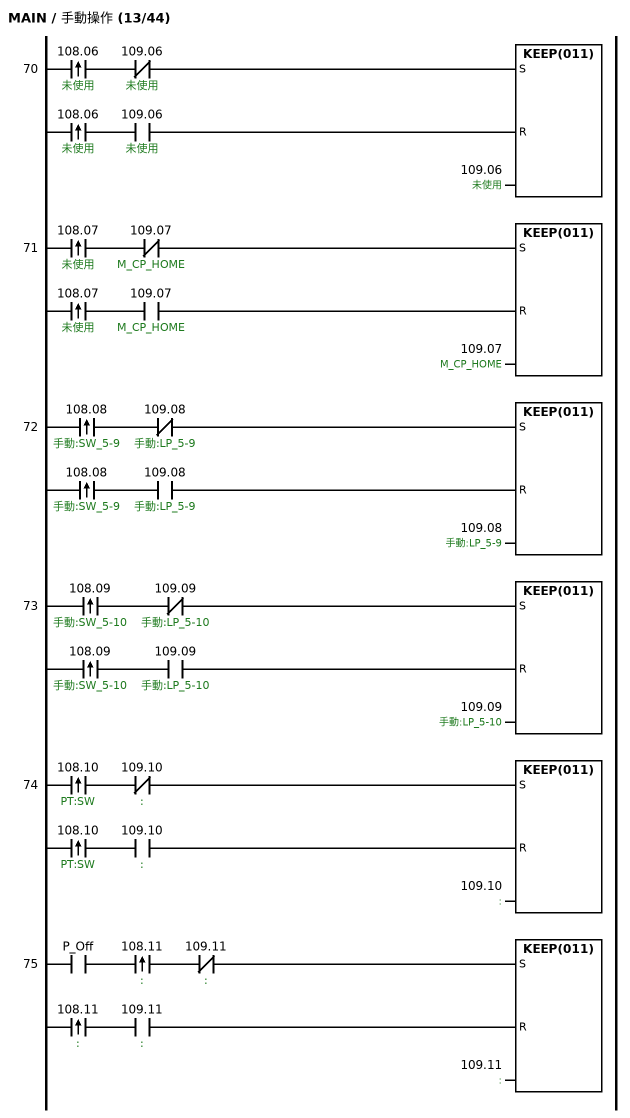
; [picture p48: MAIN / 手動操作, rungs 70-75]
; rung 70
@LD 108.06  ; 未使用
ANDNOT 109.06  ; 未使用
@LD 108.06  ; 未使用
AND 109.06  ; 未使用
KEEP(011) 109.06  ; 未使用
; rung 71
@LD 108.07  ; 未使用
ANDNOT 109.07  ; M_CP_HOME
@LD 108.07  ; 未使用
AND 109.07  ; M_CP_HOME
KEEP(011) 109.07  ; M_CP_HOME
; rung 72
@LD 108.08  ; 手動:SW_5-9
ANDNOT 109.08  ; 手動:LP_5-9
@LD 108.08  ; 手動:SW_5-9
AND 109.08  ; 手動:LP_5-9
KEEP(011) 109.08  ; 手動:LP_5-9
; rung 73
@LD 108.09  ; 手動:SW_5-10
ANDNOT 109.09  ; 手動:LP_5-10
@LD 108.09  ; 手動:SW_5-10
AND 109.09  ; 手動:LP_5-10
KEEP(011) 109.09  ; 手動:LP_5-10
; rung 74
@LD 108.10  ; PT:SW
ANDNOT 109.10  ; :
@LD 108.10  ; PT:SW
AND 109.10  ; :
KEEP(011) 109.10  ; :
; rung 75
LD P_Off
@AND 108.11  ; :
ANDNOT 109.11  ; :
@LD 108.11  ; :
AND 109.11  ; :
KEEP(011) 109.11  ; :

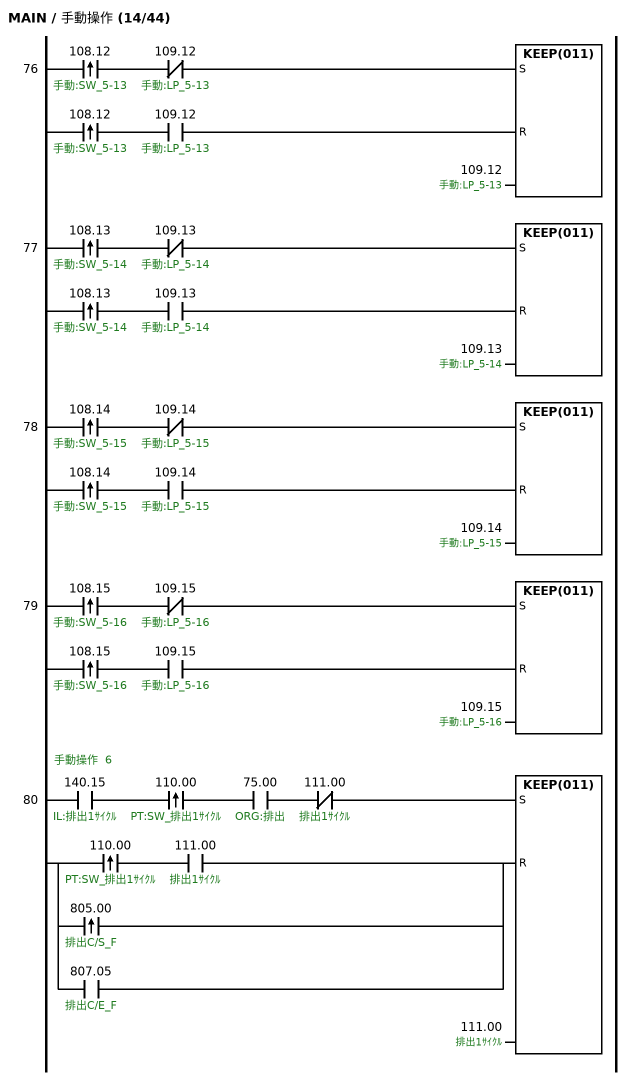
; rung 76
@LD 108.12  ; 手動:SW_5-13
ANDNOT 109.12  ; 手動:LP_5-13
@LD 108.12  ; 手動:SW_5-13
AND 109.12  ; 手動:LP_5-13
KEEP(011) 109.12  ; 手動:LP_5-13
; rung 77
@LD 108.13  ; 手動:SW_5-14
ANDNOT 109.13  ; 手動:LP_5-14
@LD 108.13  ; 手動:SW_5-14
AND 109.13  ; 手動:LP_5-14
KEEP(011) 109.13  ; 手動:LP_5-14
; rung 78
@LD 108.14  ; 手動:SW_5-15
ANDNOT 109.14  ; 手動:LP_5-15
@LD 108.14  ; 手動:SW_5-15
AND 109.14  ; 手動:LP_5-15
KEEP(011) 109.14  ; 手動:LP_5-15
; rung 79
@LD 108.15  ; 手動:SW_5-16
ANDNOT 109.15  ; 手動:LP_5-16
@LD 108.15  ; 手動:SW_5-16
AND 109.15  ; 手動:LP_5-16
KEEP(011) 109.15  ; 手動:LP_5-16
; rung 80: 手動操作  6
LD 140.15  ; IL:排出1ｻｲｸﾙ
@AND 110.00  ; PT:SW_排出1ｻｲｸﾙ
AND 75.00  ; ORG:排出
ANDNOT 111.00  ; 排出1ｻｲｸﾙ
@LD 110.00  ; PT:SW_排出1ｻｲｸﾙ
AND 111.00  ; 排出1ｻｲｸﾙ
@OR 805.00  ; 排出C/S_F
OR 807.05  ; 排出C/E_F
KEEP(011) 111.00  ; 排出1ｻｲｸﾙ

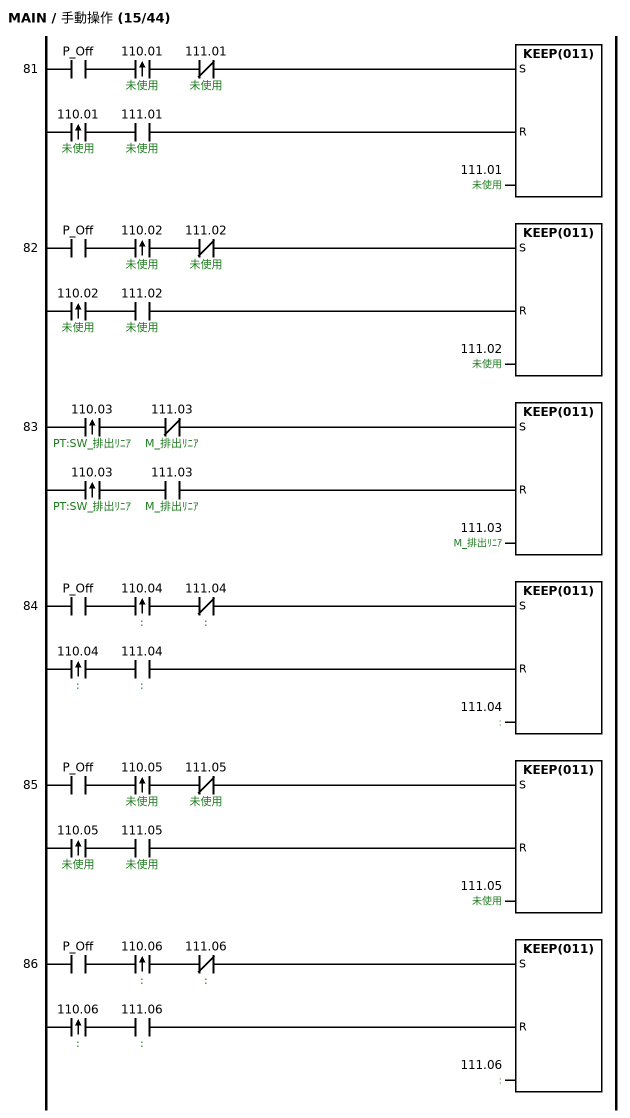
; rung 81
LD P_Off
@AND 110.01  ; 未使用
ANDNOT 111.01  ; 未使用
@LD 110.01  ; 未使用
AND 111.01  ; 未使用
KEEP(011) 111.01  ; 未使用
; rung 82
LD P_Off
@AND 110.02  ; 未使用
ANDNOT 111.02  ; 未使用
@LD 110.02  ; 未使用
AND 111.02  ; 未使用
KEEP(011) 111.02  ; 未使用
; rung 83
@LD 110.03  ; PT:SW_排出ﾘﾆｱ
ANDNOT 111.03  ; M_排出ﾘﾆｱ
@LD 110.03  ; PT:SW_排出ﾘﾆｱ
AND 111.03  ; M_排出ﾘﾆｱ
KEEP(011) 111.03  ; M_排出ﾘﾆｱ
; rung 84
LD P_Off
@AND 110.04  ; :
ANDNOT 111.04  ; :
@LD 110.04  ; :
AND 111.04  ; :
KEEP(011) 111.04  ; :
; rung 85
LD P_Off
@AND 110.05  ; 未使用
ANDNOT 111.05  ; 未使用
@LD 110.05  ; 未使用
AND 111.05  ; 未使用
KEEP(011) 111.05  ; 未使用
; rung 86
LD P_Off
@AND 110.06  ; :
ANDNOT 111.06  ; :
@LD 110.06  ; :
AND 111.06  ; :
KEEP(011) 111.06  ; :

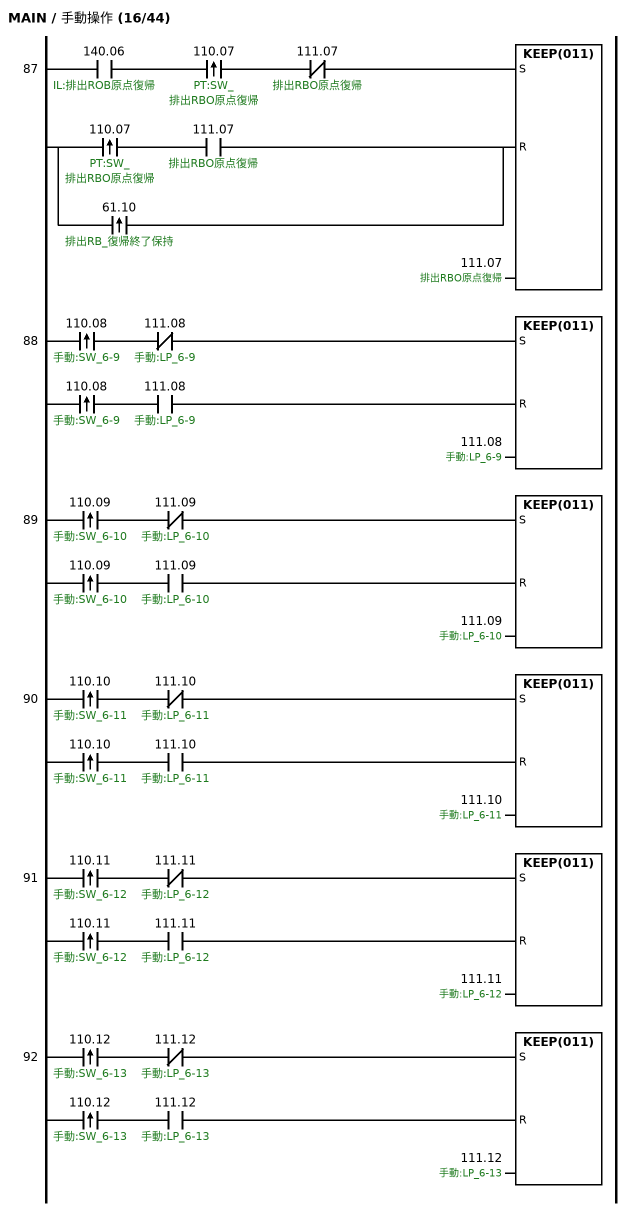
; rung 87
LD 140.06  ; IL:排出ROB原点復帰
@AND 110.07  ; PT:SW_排出RBO原点復帰
ANDNOT 111.07  ; 排出RBO原点復帰
@LD 110.07  ; PT:SW_排出RBO原点復帰
AND 111.07  ; 排出RBO原点復帰
@OR 61.10  ; 排出RB_復帰終了保持
KEEP(011) 111.07  ; 排出RBO原点復帰
; rung 88
@LD 110.08  ; 手動:SW_6-9
ANDNOT 111.08  ; 手動:LP_6-9
@LD 110.08  ; 手動:SW_6-9
AND 111.08  ; 手動:LP_6-9
KEEP(011) 111.08  ; 手動:LP_6-9
; rung 89
@LD 110.09  ; 手動:SW_6-10
ANDNOT 111.09  ; 手動:LP_6-10
@LD 110.09  ; 手動:SW_6-10
AND 111.09  ; 手動:LP_6-10
KEEP(011) 111.09  ; 手動:LP_6-10
; rung 90
@LD 110.10  ; 手動:SW_6-11
ANDNOT 111.10  ; 手動:LP_6-11
@LD 110.10  ; 手動:SW_6-11
AND 111.10  ; 手動:LP_6-11
KEEP(011) 111.10  ; 手動:LP_6-11
; rung 91
@LD 110.11  ; 手動:SW_6-12
ANDNOT 111.11  ; 手動:LP_6-12
@LD 110.11  ; 手動:SW_6-12
AND 111.11  ; 手動:LP_6-12
KEEP(011) 111.11  ; 手動:LP_6-12
; rung 92
@LD 110.12  ; 手動:SW_6-13
ANDNOT 111.12  ; 手動:LP_6-13
@LD 110.12  ; 手動:SW_6-13
AND 111.12  ; 手動:LP_6-13
KEEP(011) 111.12  ; 手動:LP_6-13

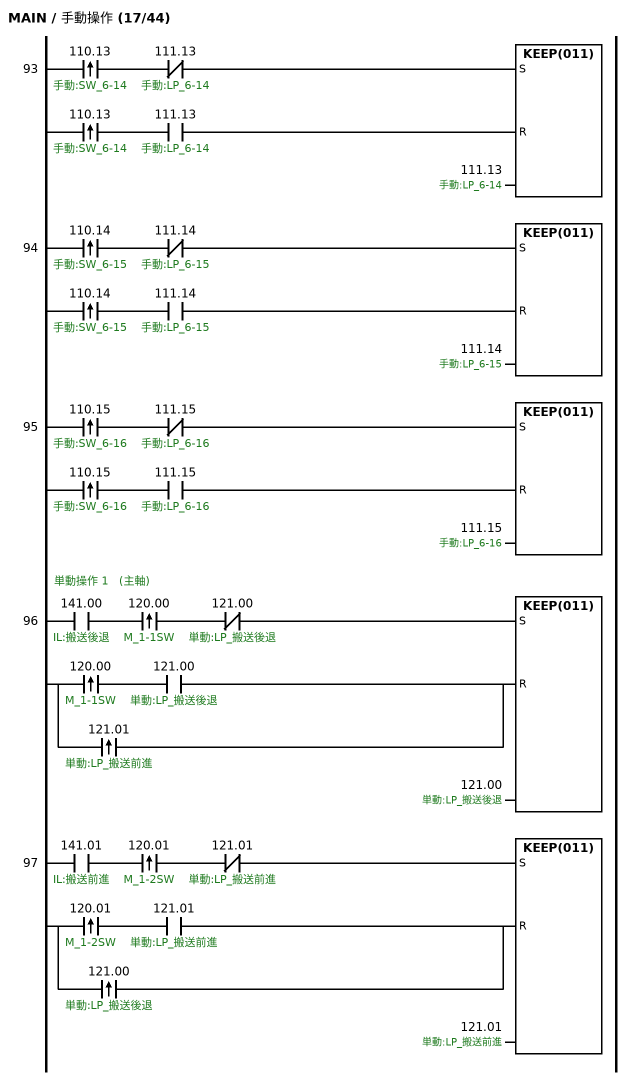
; rung 93
@LD 110.13  ; 手動:SW_6-14
ANDNOT 111.13  ; 手動:LP_6-14
@LD 110.13  ; 手動:SW_6-14
AND 111.13  ; 手動:LP_6-14
KEEP(011) 111.13  ; 手動:LP_6-14
; rung 94
@LD 110.14  ; 手動:SW_6-15
ANDNOT 111.14  ; 手動:LP_6-15
@LD 110.14  ; 手動:SW_6-15
AND 111.14  ; 手動:LP_6-15
KEEP(011) 111.14  ; 手動:LP_6-15
; rung 95
@LD 110.15  ; 手動:SW_6-16
ANDNOT 111.15  ; 手動:LP_6-16
@LD 110.15  ; 手動:SW_6-16
AND 111.15  ; 手動:LP_6-16
KEEP(011) 111.15  ; 手動:LP_6-16
; rung 96: 単動操作 1   (主軸)
LD 141.00  ; IL:搬送後退
@AND 120.00  ; M_1-1SW
ANDNOT 121.00  ; 単動:LP_搬送後退
@LD 120.00  ; M_1-1SW
AND 121.00  ; 単動:LP_搬送後退
@OR 121.01  ; 単動:LP_搬送前進
KEEP(011) 121.00  ; 単動:LP_搬送後退
; rung 97
LD 141.01  ; IL:搬送前進
@AND 120.01  ; M_1-2SW
ANDNOT 121.01  ; 単動:LP_搬送前進
@LD 120.01  ; M_1-2SW
AND 121.01  ; 単動:LP_搬送前進
@OR 121.00  ; 単動:LP_搬送後退
KEEP(011) 121.01  ; 単動:LP_搬送前進

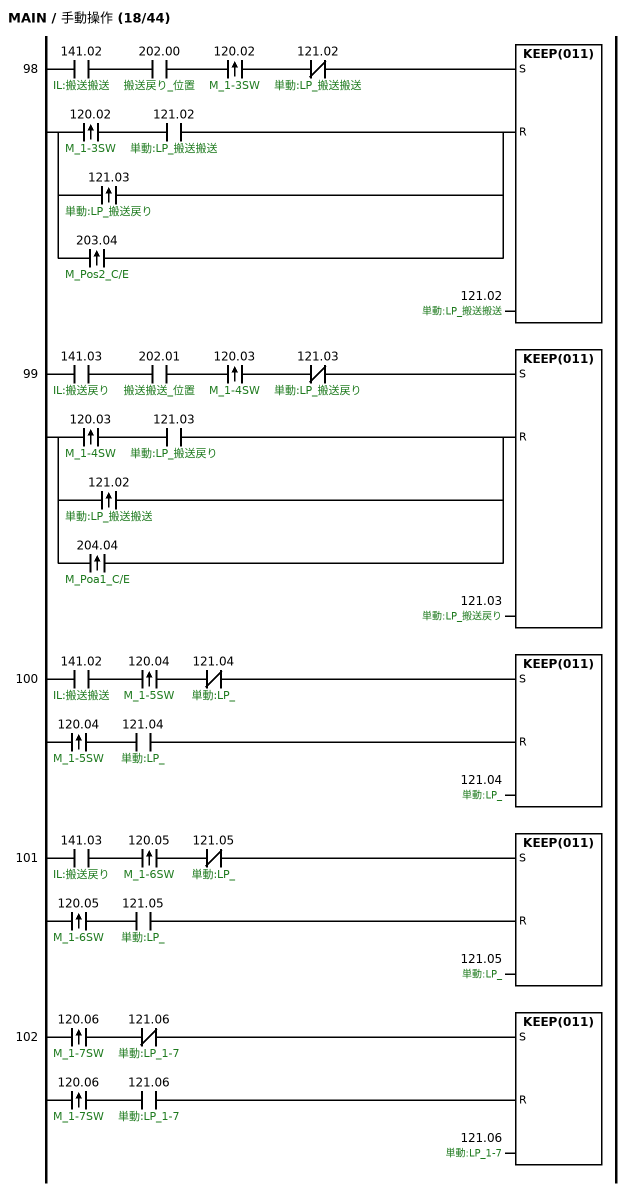
; rung 98
LD 141.02  ; IL:搬送搬送
AND 202.00  ; 搬送戻り_位置
@AND 120.02  ; M_1-3SW
ANDNOT 121.02  ; 単動:LP_搬送搬送
@LD 120.02  ; M_1-3SW
AND 121.02  ; 単動:LP_搬送搬送
@OR 121.03  ; 単動:LP_搬送戻り
@OR 203.04  ; M_Pos2_C/E
KEEP(011) 121.02  ; 単動:LP_搬送搬送
; rung 99
LD 141.03  ; IL:搬送戻り
AND 202.01  ; 搬送搬送_位置
@AND 120.03  ; M_1-4SW
ANDNOT 121.03  ; 単動:LP_搬送戻り
@LD 120.03  ; M_1-4SW
AND 121.03  ; 単動:LP_搬送戻り
@OR 121.02  ; 単動:LP_搬送搬送
@OR 204.04  ; M_Poa1_C/E
KEEP(011) 121.03  ; 単動:LP_搬送戻り
; rung 100
LD 141.02  ; IL:搬送搬送
@AND 120.04  ; M_1-5SW
ANDNOT 121.04  ; 単動:LP_
@LD 120.04  ; M_1-5SW
AND 121.04  ; 単動:LP_
KEEP(011) 121.04  ; 単動:LP_
; rung 101
LD 141.03  ; IL:搬送戻り
@AND 120.05  ; M_1-6SW
ANDNOT 121.05  ; 単動:LP_
@LD 120.05  ; M_1-6SW
AND 121.05  ; 単動:LP_
KEEP(011) 121.05  ; 単動:LP_
; rung 102
@LD 120.06  ; M_1-7SW
ANDNOT 121.06  ; 単動:LP_1-7
@LD 120.06  ; M_1-7SW
AND 121.06  ; 単動:LP_1-7
KEEP(011) 121.06  ; 単動:LP_1-7

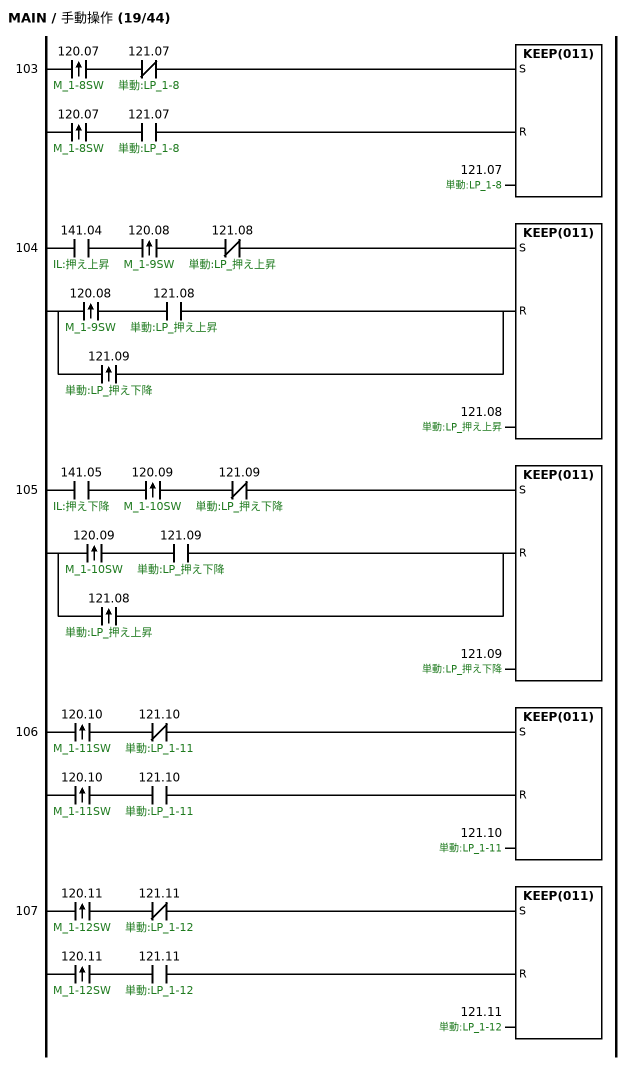
; rung 103
@LD 120.07  ; M_1-8SW
ANDNOT 121.07  ; 単動:LP_1-8
@LD 120.07  ; M_1-8SW
AND 121.07  ; 単動:LP_1-8
KEEP(011) 121.07  ; 単動:LP_1-8
; rung 104
LD 141.04  ; IL:押え上昇
@AND 120.08  ; M_1-9SW
ANDNOT 121.08  ; 単動:LP_押え上昇
@LD 120.08  ; M_1-9SW
AND 121.08  ; 単動:LP_押え上昇
@OR 121.09  ; 単動:LP_押え下降
KEEP(011) 121.08  ; 単動:LP_押え上昇
; rung 105
LD 141.05  ; IL:押え下降
@AND 120.09  ; M_1-10SW
ANDNOT 121.09  ; 単動:LP_押え下降
@LD 120.09  ; M_1-10SW
AND 121.09  ; 単動:LP_押え下降
@OR 121.08  ; 単動:LP_押え上昇
KEEP(011) 121.09  ; 単動:LP_押え下降
; rung 106
@LD 120.10  ; M_1-11SW
ANDNOT 121.10  ; 単動:LP_1-11
@LD 120.10  ; M_1-11SW
AND 121.10  ; 単動:LP_1-11
KEEP(011) 121.10  ; 単動:LP_1-11
; rung 107
@LD 120.11  ; M_1-12SW
ANDNOT 121.11  ; 単動:LP_1-12
@LD 120.11  ; M_1-12SW
AND 121.11  ; 単動:LP_1-12
KEEP(011) 121.11  ; 単動:LP_1-12

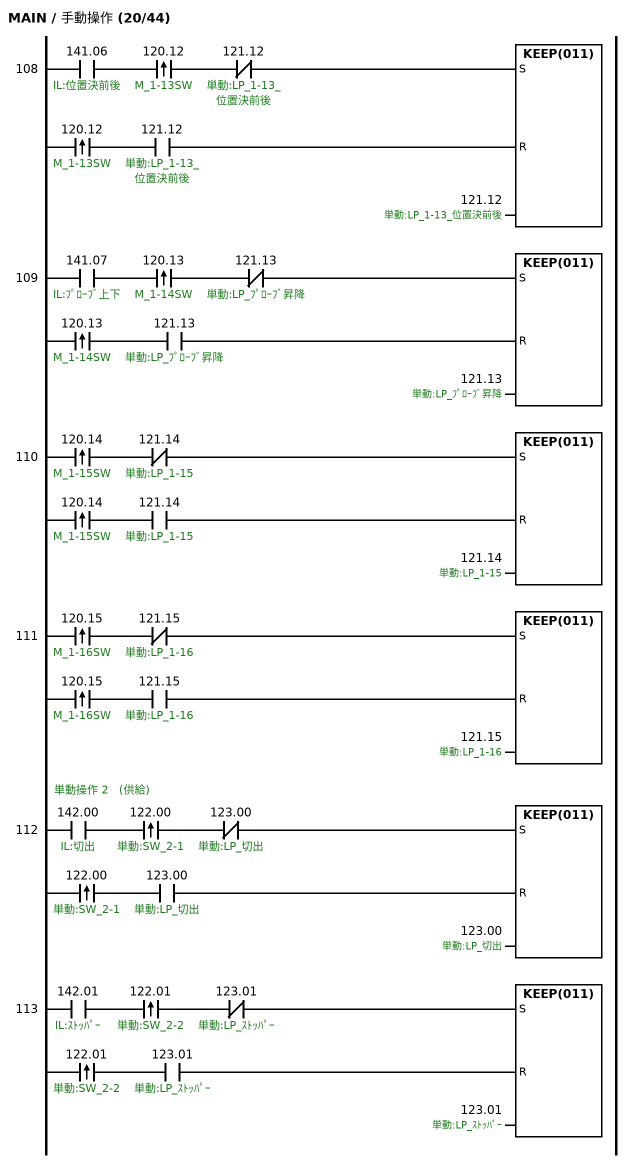
; rung 108
LD 141.06  ; IL:位置決前後
@AND 120.12  ; M_1-13SW
ANDNOT 121.12  ; 単動:LP_1-13_位置決前後
@LD 120.12  ; M_1-13SW
AND 121.12  ; 単動:LP_1-13_位置決前後
KEEP(011) 121.12  ; 単動:LP_1-13_位置決前後
; rung 109
LD 141.07  ; IL:ﾌﾟﾛｰﾌﾞ上下
@AND 120.13  ; M_1-14SW
ANDNOT 121.13  ; 単動:LP_ﾌﾟﾛｰﾌﾞ昇降
@LD 120.13  ; M_1-14SW
AND 121.13  ; 単動:LP_ﾌﾟﾛｰﾌﾞ昇降
KEEP(011) 121.13  ; 単動:LP_ﾌﾟﾛｰﾌﾞ昇降
; rung 110
@LD 120.14  ; M_1-15SW
ANDNOT 121.14  ; 単動:LP_1-15
@LD 120.14  ; M_1-15SW
AND 121.14  ; 単動:LP_1-15
KEEP(011) 121.14  ; 単動:LP_1-15
; rung 111
@LD 120.15  ; M_1-16SW
ANDNOT 121.15  ; 単動:LP_1-16
@LD 120.15  ; M_1-16SW
AND 121.15  ; 単動:LP_1-16
KEEP(011) 121.15  ; 単動:LP_1-16
; rung 112: 単動操作 2   (供給)
LD 142.00  ; IL:切出
@AND 122.00  ; 単動:SW_2-1
ANDNOT 123.00  ; 単動:LP_切出
@LD 122.00  ; 単動:SW_2-1
AND 123.00  ; 単動:LP_切出
KEEP(011) 123.00  ; 単動:LP_切出
; rung 113
LD 142.01  ; IL:ｽﾄｯﾊﾟｰ
@AND 122.01  ; 単動:SW_2-2
ANDNOT 123.01  ; 単動:LP_ｽﾄｯﾊﾟｰ
@LD 122.01  ; 単動:SW_2-2
AND 123.01  ; 単動:LP_ｽﾄｯﾊﾟｰ
KEEP(011) 123.01  ; 単動:LP_ｽﾄｯﾊﾟｰ

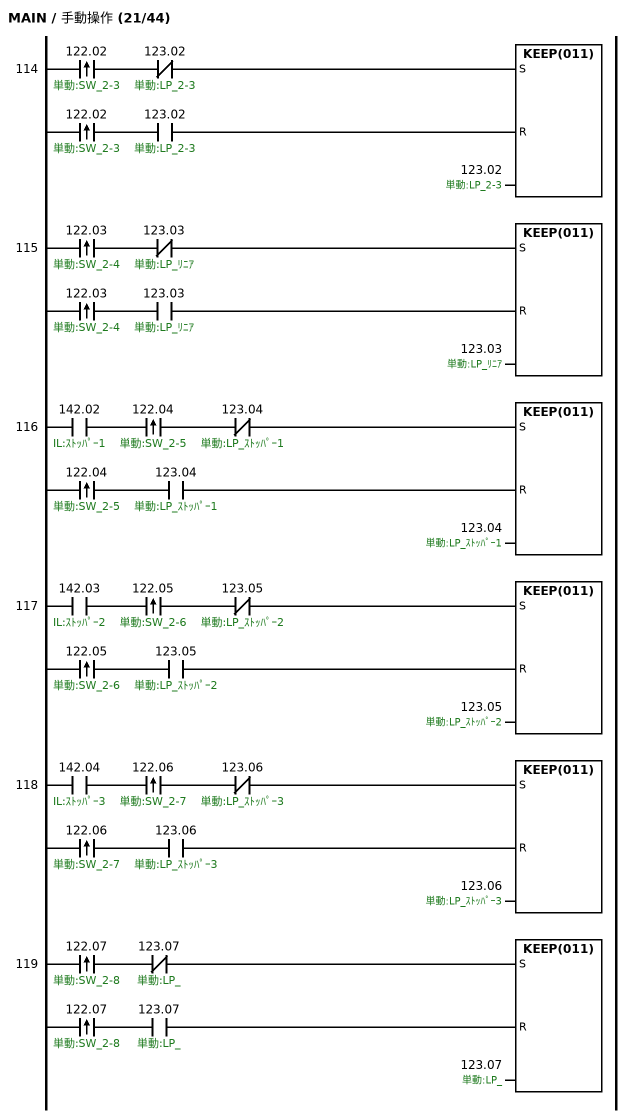
; rung 114
@LD 122.02  ; 単動:SW_2-3
ANDNOT 123.02  ; 単動:LP_2-3
@LD 122.02  ; 単動:SW_2-3
AND 123.02  ; 単動:LP_2-3
KEEP(011) 123.02  ; 単動:LP_2-3
; rung 115
@LD 122.03  ; 単動:SW_2-4
ANDNOT 123.03  ; 単動:LP_ﾘﾆｱ
@LD 122.03  ; 単動:SW_2-4
AND 123.03  ; 単動:LP_ﾘﾆｱ
KEEP(011) 123.03  ; 単動:LP_ﾘﾆｱ
; rung 116
LD 142.02  ; IL:ｽﾄｯﾊﾟｰ1
@AND 122.04  ; 単動:SW_2-5
ANDNOT 123.04  ; 単動:LP_ｽﾄｯﾊﾟｰ1
@LD 122.04  ; 単動:SW_2-5
AND 123.04  ; 単動:LP_ｽﾄｯﾊﾟｰ1
KEEP(011) 123.04  ; 単動:LP_ｽﾄｯﾊﾟｰ1
; rung 117
LD 142.03  ; IL:ｽﾄｯﾊﾟｰ2
@AND 122.05  ; 単動:SW_2-6
ANDNOT 123.05  ; 単動:LP_ｽﾄｯﾊﾟｰ2
@LD 122.05  ; 単動:SW_2-6
AND 123.05  ; 単動:LP_ｽﾄｯﾊﾟｰ2
KEEP(011) 123.05  ; 単動:LP_ｽﾄｯﾊﾟｰ2
; rung 118
LD 142.04  ; IL:ｽﾄｯﾊﾟｰ3
@AND 122.06  ; 単動:SW_2-7
ANDNOT 123.06  ; 単動:LP_ｽﾄｯﾊﾟｰ3
@LD 122.06  ; 単動:SW_2-7
AND 123.06  ; 単動:LP_ｽﾄｯﾊﾟｰ3
KEEP(011) 123.06  ; 単動:LP_ｽﾄｯﾊﾟｰ3
; rung 119
@LD 122.07  ; 単動:SW_2-8
ANDNOT 123.07  ; 単動:LP_
@LD 122.07  ; 単動:SW_2-8
AND 123.07  ; 単動:LP_
KEEP(011) 123.07  ; 単動:LP_

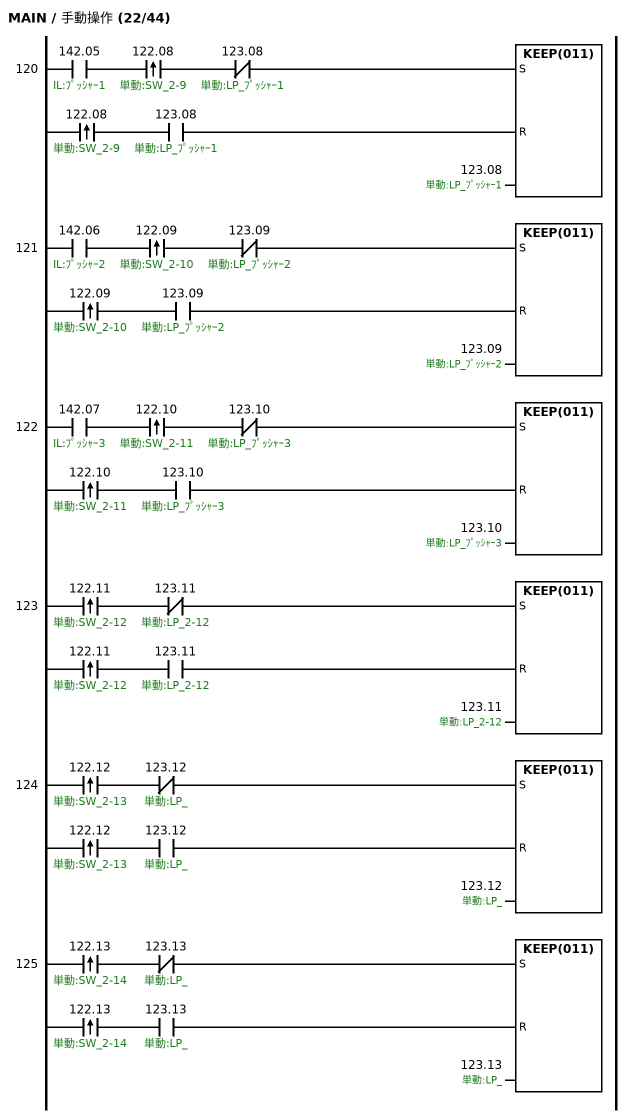
; rung 120
LD 142.05  ; IL:ﾌﾟｯｼｬｰ1
@AND 122.08  ; 単動:SW_2-9
ANDNOT 123.08  ; 単動:LP_ﾌﾟｯｼｬｰ1
@LD 122.08  ; 単動:SW_2-9
AND 123.08  ; 単動:LP_ﾌﾟｯｼｬｰ1
KEEP(011) 123.08  ; 単動:LP_ﾌﾟｯｼｬｰ1
; rung 121
LD 142.06  ; IL:ﾌﾟｯｼｬｰ2
@AND 122.09  ; 単動:SW_2-10
ANDNOT 123.09  ; 単動:LP_ﾌﾟｯｼｬｰ2
@LD 122.09  ; 単動:SW_2-10
AND 123.09  ; 単動:LP_ﾌﾟｯｼｬｰ2
KEEP(011) 123.09  ; 単動:LP_ﾌﾟｯｼｬｰ2
; rung 122
LD 142.07  ; IL:ﾌﾟｯｼｬｰ3
@AND 122.10  ; 単動:SW_2-11
ANDNOT 123.10  ; 単動:LP_ﾌﾟｯｼｬｰ3
@LD 122.10  ; 単動:SW_2-11
AND 123.10  ; 単動:LP_ﾌﾟｯｼｬｰ3
KEEP(011) 123.10  ; 単動:LP_ﾌﾟｯｼｬｰ3
; rung 123
@LD 122.11  ; 単動:SW_2-12
ANDNOT 123.11  ; 単動:LP_2-12
@LD 122.11  ; 単動:SW_2-12
AND 123.11  ; 単動:LP_2-12
KEEP(011) 123.11  ; 単動:LP_2-12
; rung 124
@LD 122.12  ; 単動:SW_2-13
ANDNOT 123.12  ; 単動:LP_
@LD 122.12  ; 単動:SW_2-13
AND 123.12  ; 単動:LP_
KEEP(011) 123.12  ; 単動:LP_
; rung 125
@LD 122.13  ; 単動:SW_2-14
ANDNOT 123.13  ; 単動:LP_
@LD 122.13  ; 単動:SW_2-14
AND 123.13  ; 単動:LP_
KEEP(011) 123.13  ; 単動:LP_

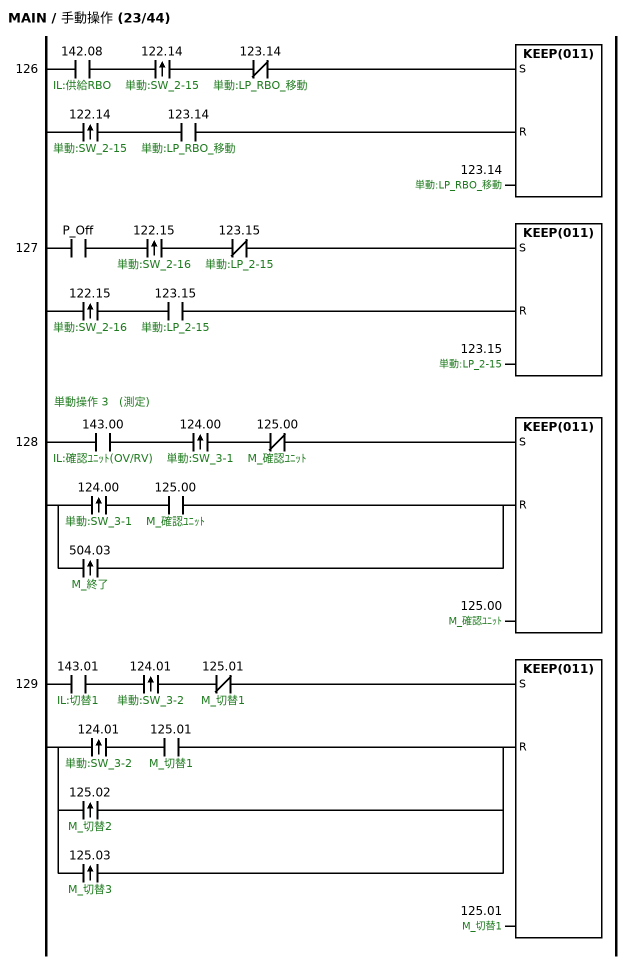
; rung 126
LD 142.08  ; IL:供給RBO
@AND 122.14  ; 単動:SW_2-15
ANDNOT 123.14  ; 単動:LP_RBO_移動
@LD 122.14  ; 単動:SW_2-15
AND 123.14  ; 単動:LP_RBO_移動
KEEP(011) 123.14  ; 単動:LP_RBO_移動
; rung 127
LD P_Off
@AND 122.15  ; 単動:SW_2-16
ANDNOT 123.15  ; 単動:LP_2-15
@LD 122.15  ; 単動:SW_2-16
AND 123.15  ; 単動:LP_2-15
KEEP(011) 123.15  ; 単動:LP_2-15
; rung 128: 単動操作 3   (測定)
LD 143.00  ; IL:確認ﾕﾆｯﾄ(OV/RV)
@AND 124.00  ; 単動:SW_3-1
ANDNOT 125.00  ; M_確認ﾕﾆｯﾄ
@LD 124.00  ; 単動:SW_3-1
AND 125.00  ; M_確認ﾕﾆｯﾄ
@OR 504.03  ; M_終了
KEEP(011) 125.00  ; M_確認ﾕﾆｯﾄ
; rung 129
LD 143.01  ; IL:切替1
@AND 124.01  ; 単動:SW_3-2
ANDNOT 125.01  ; M_切替1
@LD 124.01  ; 単動:SW_3-2
AND 125.01  ; M_切替1
@OR 125.02  ; M_切替2
@OR 125.03  ; M_切替3
KEEP(011) 125.01  ; M_切替1

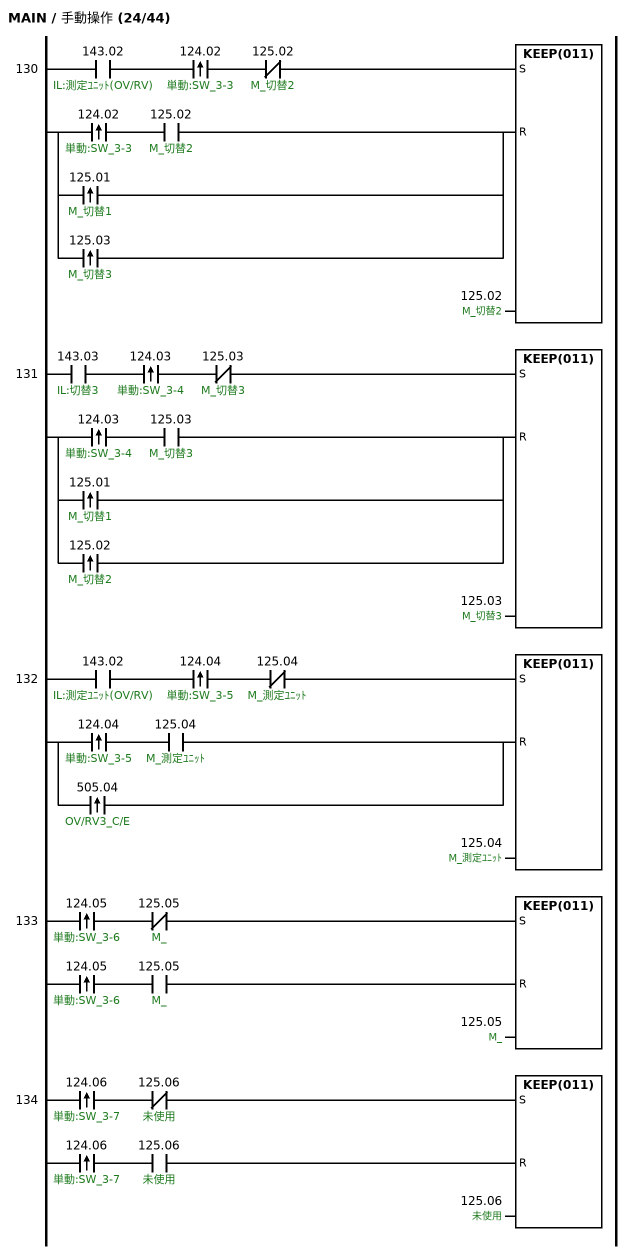
; rung 130
LD 143.02  ; IL:測定ﾕﾆｯﾄ(OV/RV)
@AND 124.02  ; 単動:SW_3-3
ANDNOT 125.02  ; M_切替2
@LD 124.02  ; 単動:SW_3-3
AND 125.02  ; M_切替2
@OR 125.01  ; M_切替1
@OR 125.03  ; M_切替3
KEEP(011) 125.02  ; M_切替2
; rung 131
LD 143.03  ; IL:切替3
@AND 124.03  ; 単動:SW_3-4
ANDNOT 125.03  ; M_切替3
@LD 124.03  ; 単動:SW_3-4
AND 125.03  ; M_切替3
@OR 125.01  ; M_切替1
@OR 125.02  ; M_切替2
KEEP(011) 125.03  ; M_切替3
; rung 132
LD 143.02  ; IL:測定ﾕﾆｯﾄ(OV/RV)
@AND 124.04  ; 単動:SW_3-5
ANDNOT 125.04  ; M_測定ﾕﾆｯﾄ
@LD 124.04  ; 単動:SW_3-5
AND 125.04  ; M_測定ﾕﾆｯﾄ
@OR 505.04  ; OV/RV3_C/E
KEEP(011) 125.04  ; M_測定ﾕﾆｯﾄ
; rung 133
@LD 124.05  ; 単動:SW_3-6
ANDNOT 125.05  ; M_
@LD 124.05  ; 単動:SW_3-6
AND 125.05  ; M_
KEEP(011) 125.05  ; M_
; rung 134
@LD 124.06  ; 単動:SW_3-7
ANDNOT 125.06  ; 未使用
@LD 124.06  ; 単動:SW_3-7
AND 125.06  ; 未使用
KEEP(011) 125.06  ; 未使用

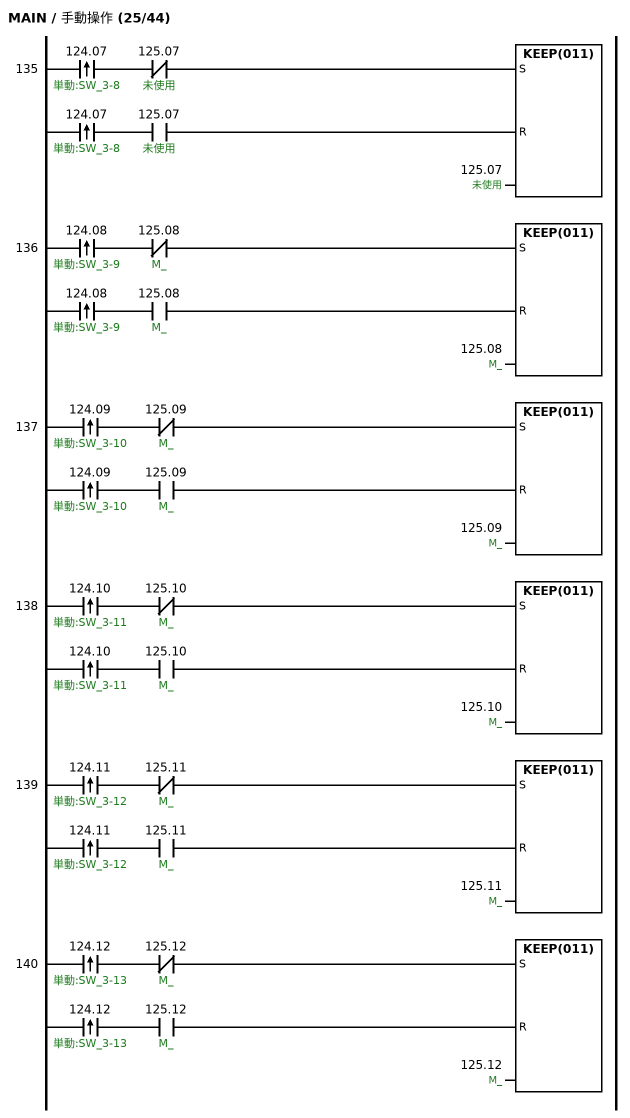
; rung 135
@LD 124.07  ; 単動:SW_3-8
ANDNOT 125.07  ; 未使用
@LD 124.07  ; 単動:SW_3-8
AND 125.07  ; 未使用
KEEP(011) 125.07  ; 未使用
; rung 136
@LD 124.08  ; 単動:SW_3-9
ANDNOT 125.08  ; M_
@LD 124.08  ; 単動:SW_3-9
AND 125.08  ; M_
KEEP(011) 125.08  ; M_
; rung 137
@LD 124.09  ; 単動:SW_3-10
ANDNOT 125.09  ; M_
@LD 124.09  ; 単動:SW_3-10
AND 125.09  ; M_
KEEP(011) 125.09  ; M_
; rung 138
@LD 124.10  ; 単動:SW_3-11
ANDNOT 125.10  ; M_
@LD 124.10  ; 単動:SW_3-11
AND 125.10  ; M_
KEEP(011) 125.10  ; M_
; rung 139
@LD 124.11  ; 単動:SW_3-12
ANDNOT 125.11  ; M_
@LD 124.11  ; 単動:SW_3-12
AND 125.11  ; M_
KEEP(011) 125.11  ; M_
; rung 140
@LD 124.12  ; 単動:SW_3-13
ANDNOT 125.12  ; M_
@LD 124.12  ; 単動:SW_3-13
AND 125.12  ; M_
KEEP(011) 125.12  ; M_

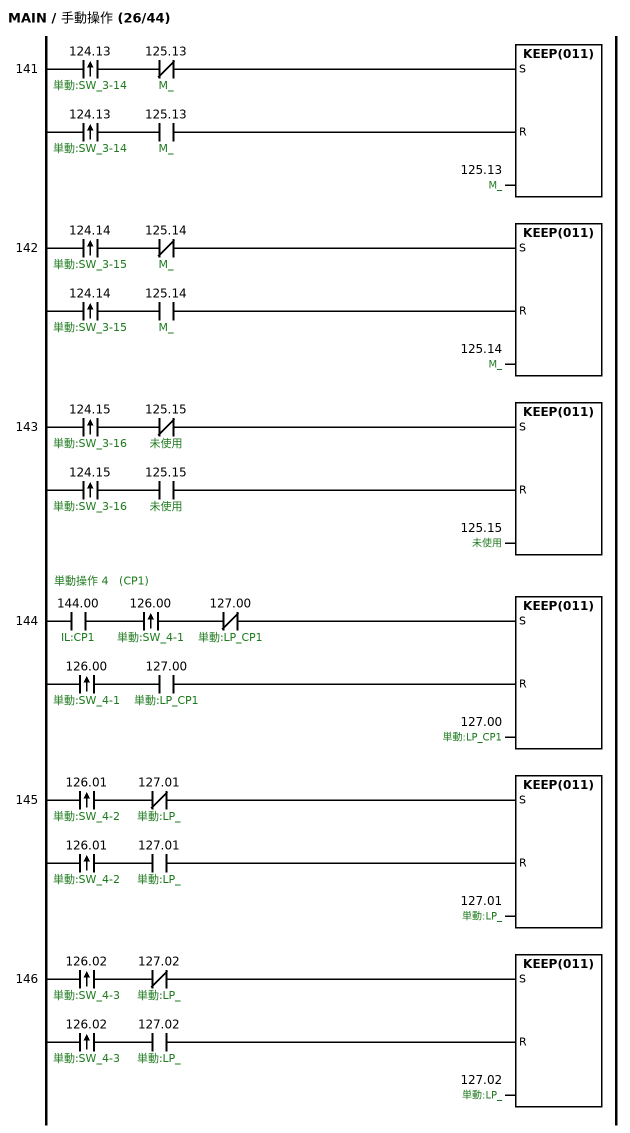
; rung 141
@LD 124.13  ; 単動:SW_3-14
ANDNOT 125.13  ; M_
@LD 124.13  ; 単動:SW_3-14
AND 125.13  ; M_
KEEP(011) 125.13  ; M_
; rung 142
@LD 124.14  ; 単動:SW_3-15
ANDNOT 125.14  ; M_
@LD 124.14  ; 単動:SW_3-15
AND 125.14  ; M_
KEEP(011) 125.14  ; M_
; rung 143
@LD 124.15  ; 単動:SW_3-16
ANDNOT 125.15  ; 未使用
@LD 124.15  ; 単動:SW_3-16
AND 125.15  ; 未使用
KEEP(011) 125.15  ; 未使用
; rung 144: 単動操作 4   (CP1)
LD 144.00  ; IL:CP1
@AND 126.00  ; 単動:SW_4-1
ANDNOT 127.00  ; 単動:LP_CP1
@LD 126.00  ; 単動:SW_4-1
AND 127.00  ; 単動:LP_CP1
KEEP(011) 127.00  ; 単動:LP_CP1
; rung 145
@LD 126.01  ; 単動:SW_4-2
ANDNOT 127.01  ; 単動:LP_
@LD 126.01  ; 単動:SW_4-2
AND 127.01  ; 単動:LP_
KEEP(011) 127.01  ; 単動:LP_
; rung 146
@LD 126.02  ; 単動:SW_4-3
ANDNOT 127.02  ; 単動:LP_
@LD 126.02  ; 単動:SW_4-3
AND 127.02  ; 単動:LP_
KEEP(011) 127.02  ; 単動:LP_

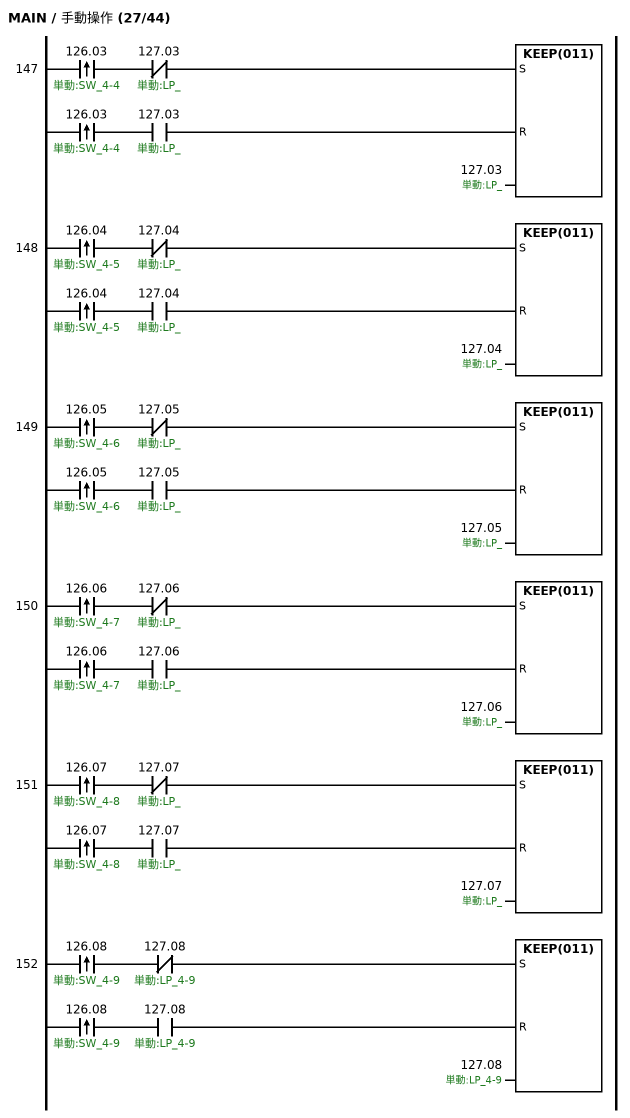
; rung 147
@LD 126.03  ; 単動:SW_4-4
ANDNOT 127.03  ; 単動:LP_
@LD 126.03  ; 単動:SW_4-4
AND 127.03  ; 単動:LP_
KEEP(011) 127.03  ; 単動:LP_
; rung 148
@LD 126.04  ; 単動:SW_4-5
ANDNOT 127.04  ; 単動:LP_
@LD 126.04  ; 単動:SW_4-5
AND 127.04  ; 単動:LP_
KEEP(011) 127.04  ; 単動:LP_
; rung 149
@LD 126.05  ; 単動:SW_4-6
ANDNOT 127.05  ; 単動:LP_
@LD 126.05  ; 単動:SW_4-6
AND 127.05  ; 単動:LP_
KEEP(011) 127.05  ; 単動:LP_
; rung 150
@LD 126.06  ; 単動:SW_4-7
ANDNOT 127.06  ; 単動:LP_
@LD 126.06  ; 単動:SW_4-7
AND 127.06  ; 単動:LP_
KEEP(011) 127.06  ; 単動:LP_
; rung 151
@LD 126.07  ; 単動:SW_4-8
ANDNOT 127.07  ; 単動:LP_
@LD 126.07  ; 単動:SW_4-8
AND 127.07  ; 単動:LP_
KEEP(011) 127.07  ; 単動:LP_
; rung 152
@LD 126.08  ; 単動:SW_4-9
ANDNOT 127.08  ; 単動:LP_4-9
@LD 126.08  ; 単動:SW_4-9
AND 127.08  ; 単動:LP_4-9
KEEP(011) 127.08  ; 単動:LP_4-9

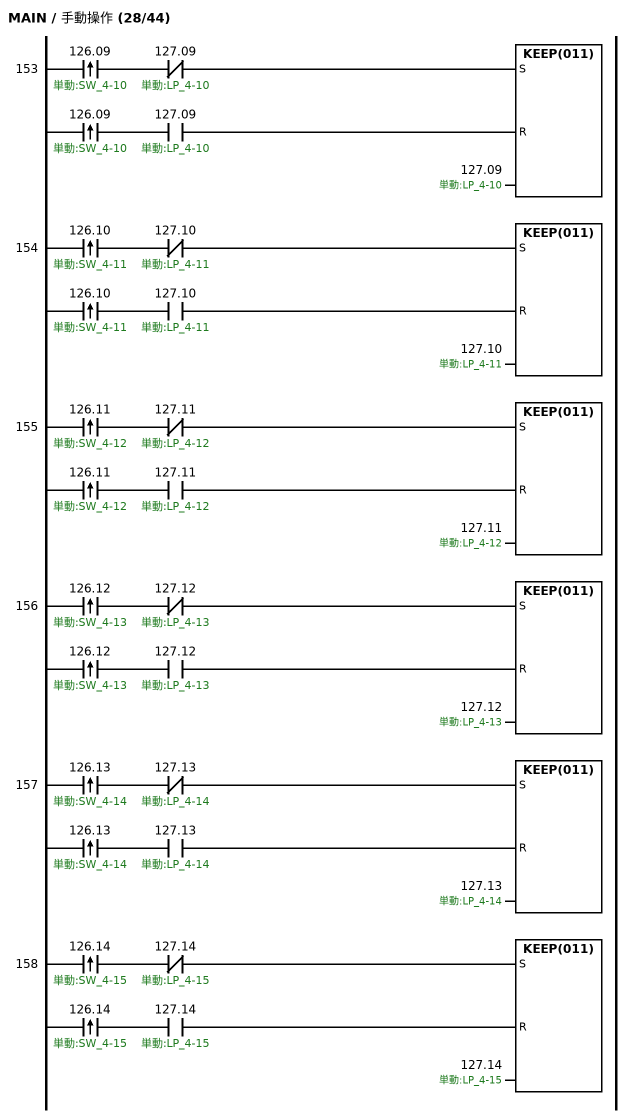
; rung 153
@LD 126.09  ; 単動:SW_4-10
ANDNOT 127.09  ; 単動:LP_4-10
@LD 126.09  ; 単動:SW_4-10
AND 127.09  ; 単動:LP_4-10
KEEP(011) 127.09  ; 単動:LP_4-10
; rung 154
@LD 126.10  ; 単動:SW_4-11
ANDNOT 127.10  ; 単動:LP_4-11
@LD 126.10  ; 単動:SW_4-11
AND 127.10  ; 単動:LP_4-11
KEEP(011) 127.10  ; 単動:LP_4-11
; rung 155
@LD 126.11  ; 単動:SW_4-12
ANDNOT 127.11  ; 単動:LP_4-12
@LD 126.11  ; 単動:SW_4-12
AND 127.11  ; 単動:LP_4-12
KEEP(011) 127.11  ; 単動:LP_4-12
; rung 156
@LD 126.12  ; 単動:SW_4-13
ANDNOT 127.12  ; 単動:LP_4-13
@LD 126.12  ; 単動:SW_4-13
AND 127.12  ; 単動:LP_4-13
KEEP(011) 127.12  ; 単動:LP_4-13
; rung 157
@LD 126.13  ; 単動:SW_4-14
ANDNOT 127.13  ; 単動:LP_4-14
@LD 126.13  ; 単動:SW_4-14
AND 127.13  ; 単動:LP_4-14
KEEP(011) 127.13  ; 単動:LP_4-14
; rung 158
@LD 126.14  ; 単動:SW_4-15
ANDNOT 127.14  ; 単動:LP_4-15
@LD 126.14  ; 単動:SW_4-15
AND 127.14  ; 単動:LP_4-15
KEEP(011) 127.14  ; 単動:LP_4-15

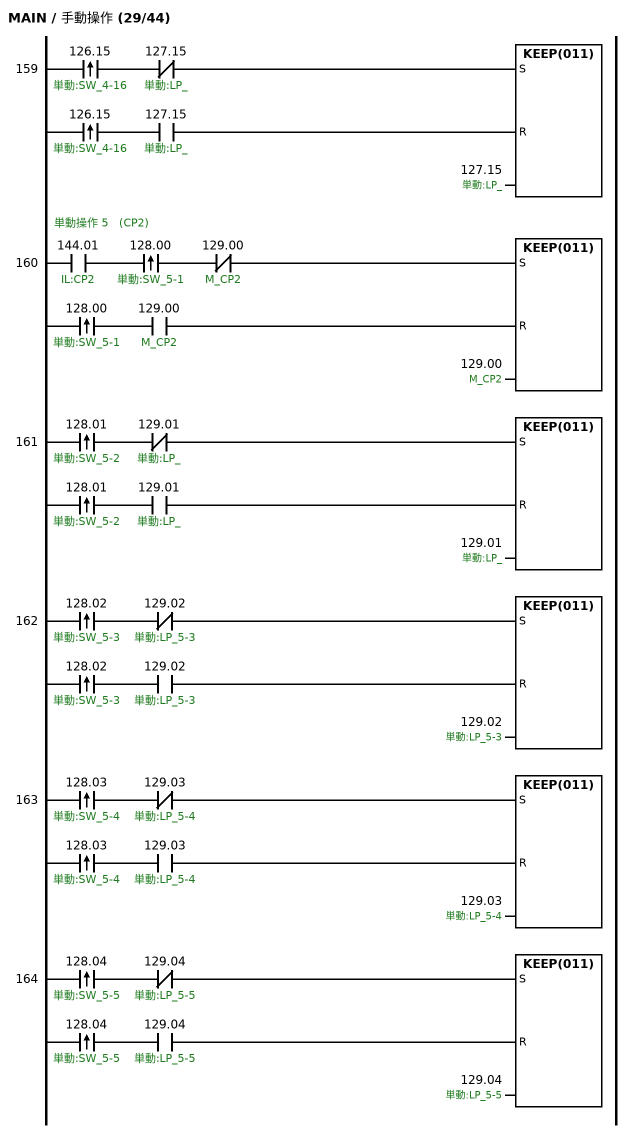
; rung 159
@LD 126.15  ; 単動:SW_4-16
ANDNOT 127.15  ; 単動:LP_
@LD 126.15  ; 単動:SW_4-16
AND 127.15  ; 単動:LP_
KEEP(011) 127.15  ; 単動:LP_
; rung 160: 単動操作 5   (CP2)
LD 144.01  ; IL:CP2
@AND 128.00  ; 単動:SW_5-1
ANDNOT 129.00  ; M_CP2
@LD 128.00  ; 単動:SW_5-1
AND 129.00  ; M_CP2
KEEP(011) 129.00  ; M_CP2
; rung 161
@LD 128.01  ; 単動:SW_5-2
ANDNOT 129.01  ; 単動:LP_
@LD 128.01  ; 単動:SW_5-2
AND 129.01  ; 単動:LP_
KEEP(011) 129.01  ; 単動:LP_
; rung 162
@LD 128.02  ; 単動:SW_5-3
ANDNOT 129.02  ; 単動:LP_5-3
@LD 128.02  ; 単動:SW_5-3
AND 129.02  ; 単動:LP_5-3
KEEP(011) 129.02  ; 単動:LP_5-3
; rung 163
@LD 128.03  ; 単動:SW_5-4
ANDNOT 129.03  ; 単動:LP_5-4
@LD 128.03  ; 単動:SW_5-4
AND 129.03  ; 単動:LP_5-4
KEEP(011) 129.03  ; 単動:LP_5-4
; rung 164
@LD 128.04  ; 単動:SW_5-5
ANDNOT 129.04  ; 単動:LP_5-5
@LD 128.04  ; 単動:SW_5-5
AND 129.04  ; 単動:LP_5-5
KEEP(011) 129.04  ; 単動:LP_5-5

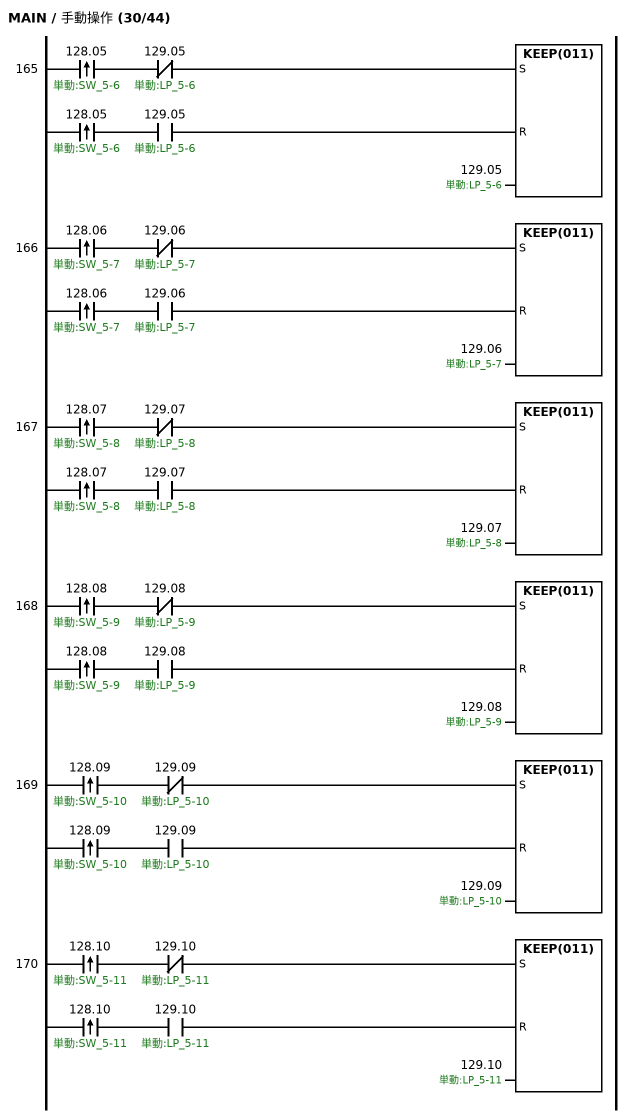
; rung 165
@LD 128.05  ; 単動:SW_5-6
ANDNOT 129.05  ; 単動:LP_5-6
@LD 128.05  ; 単動:SW_5-6
AND 129.05  ; 単動:LP_5-6
KEEP(011) 129.05  ; 単動:LP_5-6
; rung 166
@LD 128.06  ; 単動:SW_5-7
ANDNOT 129.06  ; 単動:LP_5-7
@LD 128.06  ; 単動:SW_5-7
AND 129.06  ; 単動:LP_5-7
KEEP(011) 129.06  ; 単動:LP_5-7
; rung 167
@LD 128.07  ; 単動:SW_5-8
ANDNOT 129.07  ; 単動:LP_5-8
@LD 128.07  ; 単動:SW_5-8
AND 129.07  ; 単動:LP_5-8
KEEP(011) 129.07  ; 単動:LP_5-8
; rung 168
@LD 128.08  ; 単動:SW_5-9
ANDNOT 129.08  ; 単動:LP_5-9
@LD 128.08  ; 単動:SW_5-9
AND 129.08  ; 単動:LP_5-9
KEEP(011) 129.08  ; 単動:LP_5-9
; rung 169
@LD 128.09  ; 単動:SW_5-10
ANDNOT 129.09  ; 単動:LP_5-10
@LD 128.09  ; 単動:SW_5-10
AND 129.09  ; 単動:LP_5-10
KEEP(011) 129.09  ; 単動:LP_5-10
; rung 170
@LD 128.10  ; 単動:SW_5-11
ANDNOT 129.10  ; 単動:LP_5-11
@LD 128.10  ; 単動:SW_5-11
AND 129.10  ; 単動:LP_5-11
KEEP(011) 129.10  ; 単動:LP_5-11

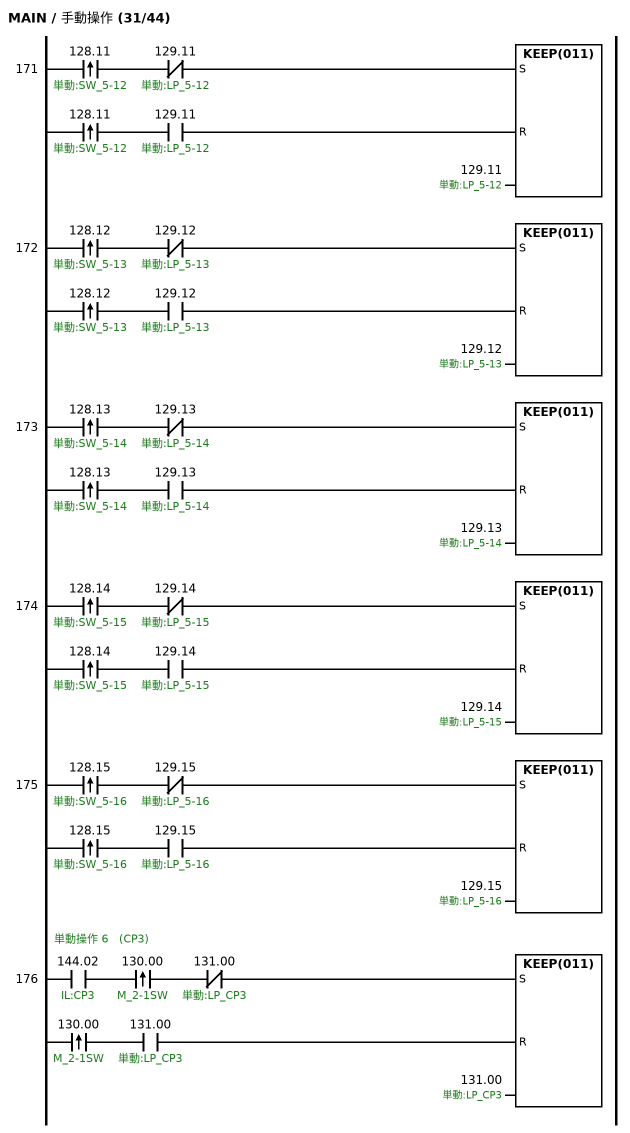
; rung 171
@LD 128.11  ; 単動:SW_5-12
ANDNOT 129.11  ; 単動:LP_5-12
@LD 128.11  ; 単動:SW_5-12
AND 129.11  ; 単動:LP_5-12
KEEP(011) 129.11  ; 単動:LP_5-12
; rung 172
@LD 128.12  ; 単動:SW_5-13
ANDNOT 129.12  ; 単動:LP_5-13
@LD 128.12  ; 単動:SW_5-13
AND 129.12  ; 単動:LP_5-13
KEEP(011) 129.12  ; 単動:LP_5-13
; rung 173
@LD 128.13  ; 単動:SW_5-14
ANDNOT 129.13  ; 単動:LP_5-14
@LD 128.13  ; 単動:SW_5-14
AND 129.13  ; 単動:LP_5-14
KEEP(011) 129.13  ; 単動:LP_5-14
; rung 174
@LD 128.14  ; 単動:SW_5-15
ANDNOT 129.14  ; 単動:LP_5-15
@LD 128.14  ; 単動:SW_5-15
AND 129.14  ; 単動:LP_5-15
KEEP(011) 129.14  ; 単動:LP_5-15
; rung 175
@LD 128.15  ; 単動:SW_5-16
ANDNOT 129.15  ; 単動:LP_5-16
@LD 128.15  ; 単動:SW_5-16
AND 129.15  ; 単動:LP_5-16
KEEP(011) 129.15  ; 単動:LP_5-16
; rung 176: 単動操作 6   (CP3)
LD 144.02  ; IL:CP3
@AND 130.00  ; M_2-1SW
ANDNOT 131.00  ; 単動:LP_CP3
@LD 130.00  ; M_2-1SW
AND 131.00  ; 単動:LP_CP3
KEEP(011) 131.00  ; 単動:LP_CP3

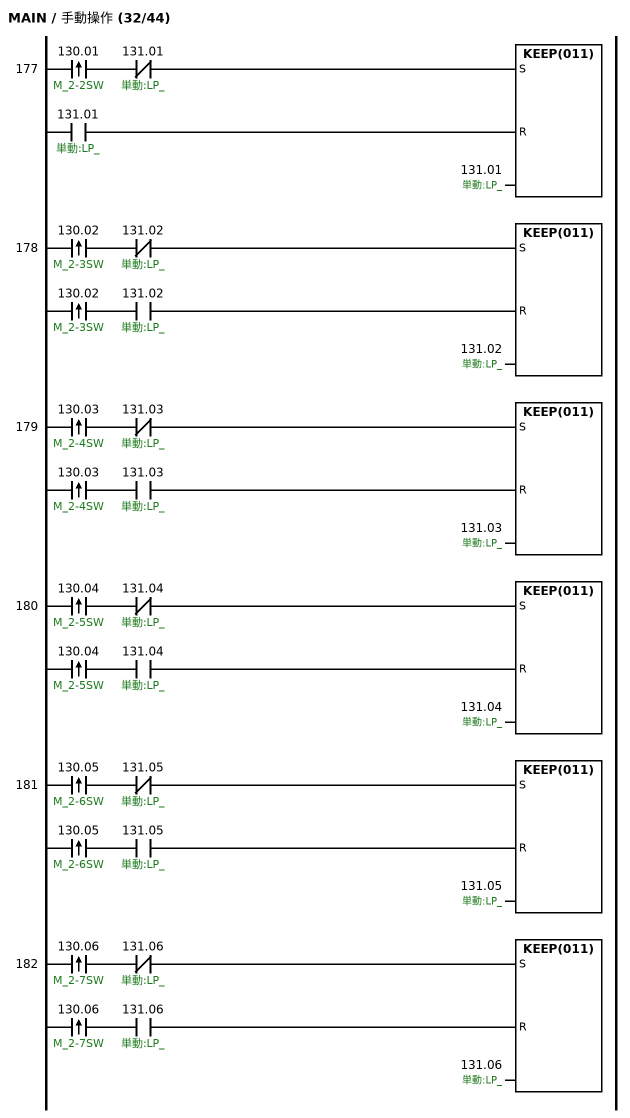
; rung 177
@LD 130.01  ; M_2-2SW
ANDNOT 131.01  ; 単動:LP_
LD 131.01  ; 単動:LP_
KEEP(011) 131.01  ; 単動:LP_
; rung 178
@LD 130.02  ; M_2-3SW
ANDNOT 131.02  ; 単動:LP_
@LD 130.02  ; M_2-3SW
AND 131.02  ; 単動:LP_
KEEP(011) 131.02  ; 単動:LP_
; rung 179
@LD 130.03  ; M_2-4SW
ANDNOT 131.03  ; 単動:LP_
@LD 130.03  ; M_2-4SW
AND 131.03  ; 単動:LP_
KEEP(011) 131.03  ; 単動:LP_
; rung 180
@LD 130.04  ; M_2-5SW
ANDNOT 131.04  ; 単動:LP_
@LD 130.04  ; M_2-5SW
AND 131.04  ; 単動:LP_
KEEP(011) 131.04  ; 単動:LP_
; rung 181
@LD 130.05  ; M_2-6SW
ANDNOT 131.05  ; 単動:LP_
@LD 130.05  ; M_2-6SW
AND 131.05  ; 単動:LP_
KEEP(011) 131.05  ; 単動:LP_
; rung 182
@LD 130.06  ; M_2-7SW
ANDNOT 131.06  ; 単動:LP_
@LD 130.06  ; M_2-7SW
AND 131.06  ; 単動:LP_
KEEP(011) 131.06  ; 単動:LP_

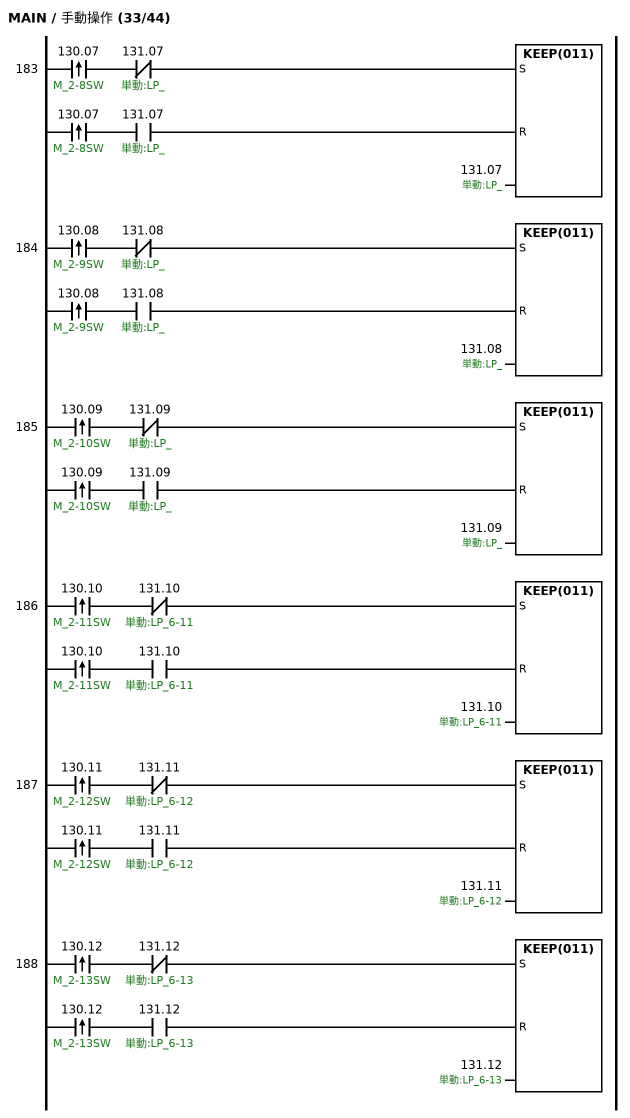
; rung 183
@LD 130.07  ; M_2-8SW
ANDNOT 131.07  ; 単動:LP_
@LD 130.07  ; M_2-8SW
AND 131.07  ; 単動:LP_
KEEP(011) 131.07  ; 単動:LP_
; rung 184
@LD 130.08  ; M_2-9SW
ANDNOT 131.08  ; 単動:LP_
@LD 130.08  ; M_2-9SW
AND 131.08  ; 単動:LP_
KEEP(011) 131.08  ; 単動:LP_
; rung 185
@LD 130.09  ; M_2-10SW
ANDNOT 131.09  ; 単動:LP_
@LD 130.09  ; M_2-10SW
AND 131.09  ; 単動:LP_
KEEP(011) 131.09  ; 単動:LP_
; rung 186
@LD 130.10  ; M_2-11SW
ANDNOT 131.10  ; 単動:LP_6-11
@LD 130.10  ; M_2-11SW
AND 131.10  ; 単動:LP_6-11
KEEP(011) 131.10  ; 単動:LP_6-11
; rung 187
@LD 130.11  ; M_2-12SW
ANDNOT 131.11  ; 単動:LP_6-12
@LD 130.11  ; M_2-12SW
AND 131.11  ; 単動:LP_6-12
KEEP(011) 131.11  ; 単動:LP_6-12
; rung 188
@LD 130.12  ; M_2-13SW
ANDNOT 131.12  ; 単動:LP_6-13
@LD 130.12  ; M_2-13SW
AND 131.12  ; 単動:LP_6-13
KEEP(011) 131.12  ; 単動:LP_6-13

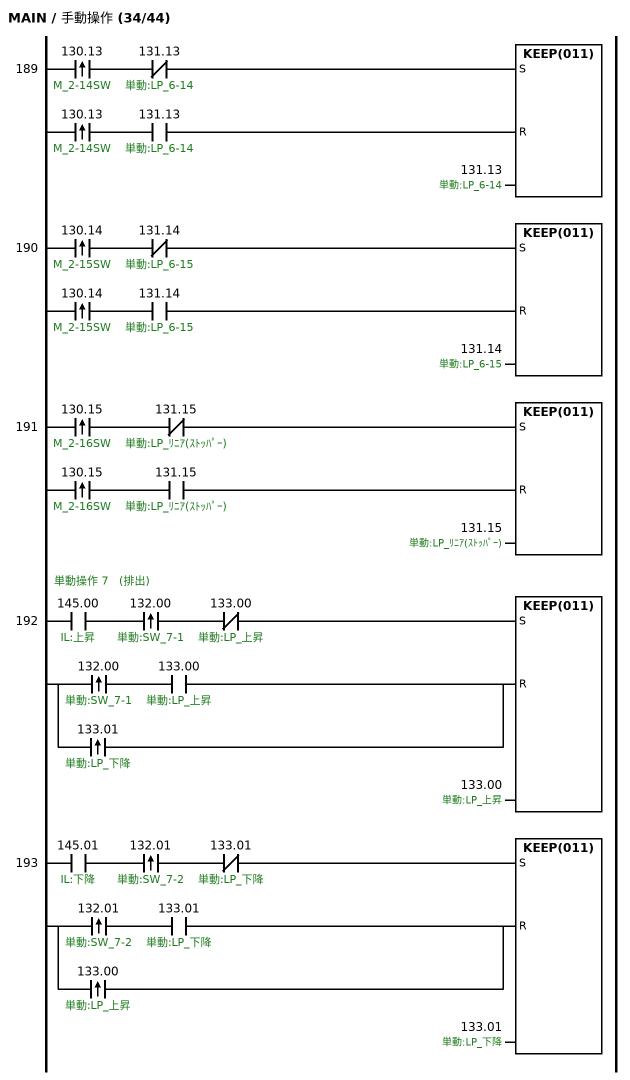
; rung 189
@LD 130.13  ; M_2-14SW
ANDNOT 131.13  ; 単動:LP_6-14
@LD 130.13  ; M_2-14SW
AND 131.13  ; 単動:LP_6-14
KEEP(011) 131.13  ; 単動:LP_6-14
; rung 190
@LD 130.14  ; M_2-15SW
ANDNOT 131.14  ; 単動:LP_6-15
@LD 130.14  ; M_2-15SW
AND 131.14  ; 単動:LP_6-15
KEEP(011) 131.14  ; 単動:LP_6-15
; rung 191
@LD 130.15  ; M_2-16SW
ANDNOT 131.15  ; 単動:LP_ﾘﾆｱ(ｽﾄｯﾊﾟｰ)
@LD 130.15  ; M_2-16SW
AND 131.15  ; 単動:LP_ﾘﾆｱ(ｽﾄｯﾊﾟｰ)
KEEP(011) 131.15  ; 単動:LP_ﾘﾆｱ(ｽﾄｯﾊﾟｰ)
; rung 192: 単動操作 7   (排出)
LD 145.00  ; IL:上昇
@AND 132.00  ; 単動:SW_7-1
ANDNOT 133.00  ; 単動:LP_上昇
@LD 132.00  ; 単動:SW_7-1
AND 133.00  ; 単動:LP_上昇
@OR 133.01  ; 単動:LP_下降
KEEP(011) 133.00  ; 単動:LP_上昇
; rung 193
LD 145.01  ; IL:下降
@AND 132.01  ; 単動:SW_7-2
ANDNOT 133.01  ; 単動:LP_下降
@LD 132.01  ; 単動:SW_7-2
AND 133.01  ; 単動:LP_下降
@OR 133.00  ; 単動:LP_上昇
KEEP(011) 133.01  ; 単動:LP_下降

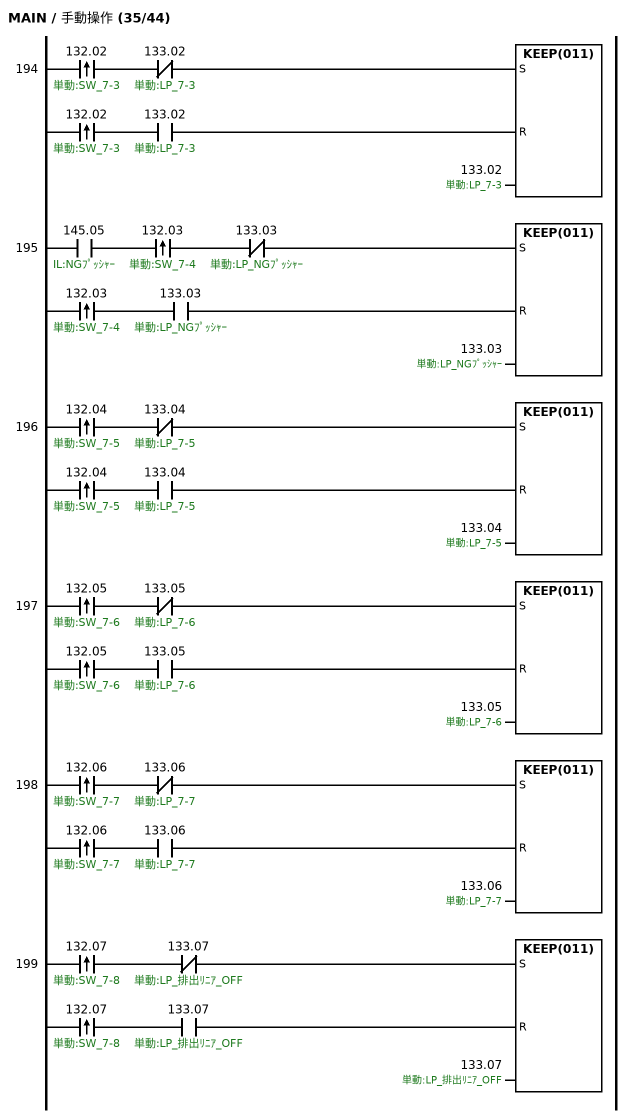
; rung 194
@LD 132.02  ; 単動:SW_7-3
ANDNOT 133.02  ; 単動:LP_7-3
@LD 132.02  ; 単動:SW_7-3
AND 133.02  ; 単動:LP_7-3
KEEP(011) 133.02  ; 単動:LP_7-3
; rung 195
LD 145.05  ; IL:NGﾌﾟｯｼｬｰ
@AND 132.03  ; 単動:SW_7-4
ANDNOT 133.03  ; 単動:LP_NGﾌﾟｯｼｬｰ
@LD 132.03  ; 単動:SW_7-4
AND 133.03  ; 単動:LP_NGﾌﾟｯｼｬｰ
KEEP(011) 133.03  ; 単動:LP_NGﾌﾟｯｼｬｰ
; rung 196
@LD 132.04  ; 単動:SW_7-5
ANDNOT 133.04  ; 単動:LP_7-5
@LD 132.04  ; 単動:SW_7-5
AND 133.04  ; 単動:LP_7-5
KEEP(011) 133.04  ; 単動:LP_7-5
; rung 197
@LD 132.05  ; 単動:SW_7-6
ANDNOT 133.05  ; 単動:LP_7-6
@LD 132.05  ; 単動:SW_7-6
AND 133.05  ; 単動:LP_7-6
KEEP(011) 133.05  ; 単動:LP_7-6
; rung 198
@LD 132.06  ; 単動:SW_7-7
ANDNOT 133.06  ; 単動:LP_7-7
@LD 132.06  ; 単動:SW_7-7
AND 133.06  ; 単動:LP_7-7
KEEP(011) 133.06  ; 単動:LP_7-7
; rung 199
@LD 132.07  ; 単動:SW_7-8
ANDNOT 133.07  ; 単動:LP_排出ﾘﾆｱ_OFF
@LD 132.07  ; 単動:SW_7-8
AND 133.07  ; 単動:LP_排出ﾘﾆｱ_OFF
KEEP(011) 133.07  ; 単動:LP_排出ﾘﾆｱ_OFF

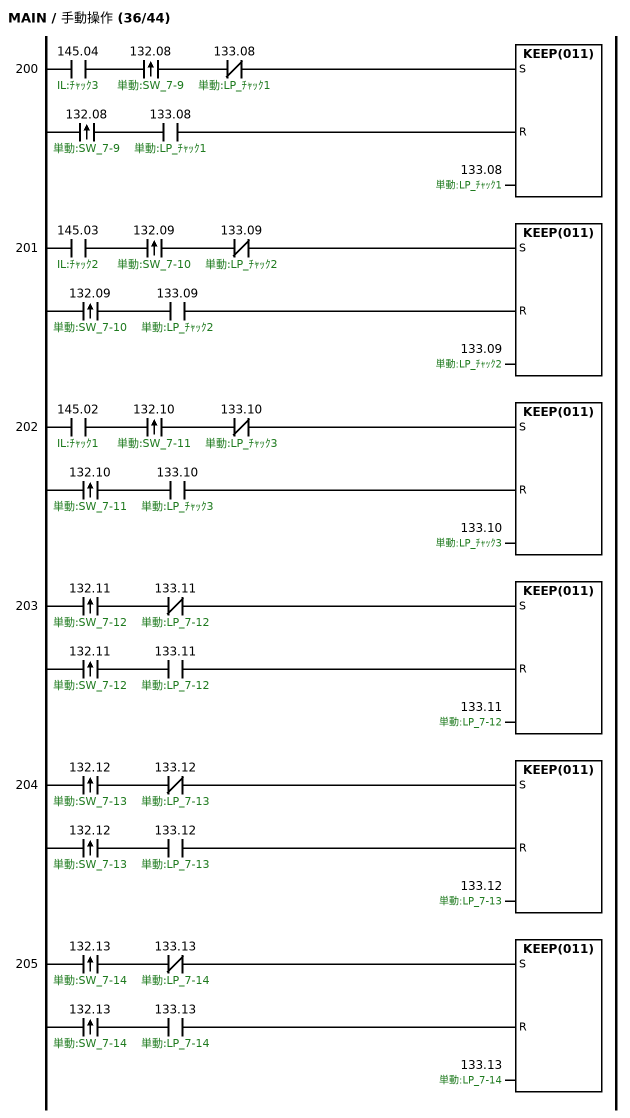
; rung 200
LD 145.04  ; IL:ﾁｬｯｸ3
@AND 132.08  ; 単動:SW_7-9
ANDNOT 133.08  ; 単動:LP_ﾁｬｯｸ1
@LD 132.08  ; 単動:SW_7-9
AND 133.08  ; 単動:LP_ﾁｬｯｸ1
KEEP(011) 133.08  ; 単動:LP_ﾁｬｯｸ1
; rung 201
LD 145.03  ; IL:ﾁｬｯｸ2
@AND 132.09  ; 単動:SW_7-10
ANDNOT 133.09  ; 単動:LP_ﾁｬｯｸ2
@LD 132.09  ; 単動:SW_7-10
AND 133.09  ; 単動:LP_ﾁｬｯｸ2
KEEP(011) 133.09  ; 単動:LP_ﾁｬｯｸ2
; rung 202
LD 145.02  ; IL:ﾁｬｯｸ1
@AND 132.10  ; 単動:SW_7-11
ANDNOT 133.10  ; 単動:LP_ﾁｬｯｸ3
@LD 132.10  ; 単動:SW_7-11
AND 133.10  ; 単動:LP_ﾁｬｯｸ3
KEEP(011) 133.10  ; 単動:LP_ﾁｬｯｸ3
; rung 203
@LD 132.11  ; 単動:SW_7-12
ANDNOT 133.11  ; 単動:LP_7-12
@LD 132.11  ; 単動:SW_7-12
AND 133.11  ; 単動:LP_7-12
KEEP(011) 133.11  ; 単動:LP_7-12
; rung 204
@LD 132.12  ; 単動:SW_7-13
ANDNOT 133.12  ; 単動:LP_7-13
@LD 132.12  ; 単動:SW_7-13
AND 133.12  ; 単動:LP_7-13
KEEP(011) 133.12  ; 単動:LP_7-13
; rung 205
@LD 132.13  ; 単動:SW_7-14
ANDNOT 133.13  ; 単動:LP_7-14
@LD 132.13  ; 単動:SW_7-14
AND 133.13  ; 単動:LP_7-14
KEEP(011) 133.13  ; 単動:LP_7-14

